FUNCTION F_ParToCsvLine : T_MaxString // convert parameter into csv string (default UDt_Parameter setup)
VAR_INPUT
	stParameter : Udt_Parameter ; 
	nColumn		: UDINT ;
END_VAR
VAR
	sTempString : T_MaxString;
	sTempCsvField : T_MaxString;
END_VAR

CASE nColumn OF 
	0: // number
		sTempString := UDINT_TO_STRING(stParameter.nNumber);
	1: // name
		sTempString := stParameter.sName;
	2: // Type
		sTempString := stParameter.sType;
	3: // discription
		sTempString := stParameter.sDiscription;
	4: // factory
		sTempString := LREAL_TO_STRING(stParameter.fFactory);
	5: // maximum
		sTempString := LREAL_TO_STRING(stParameter.fMaximum);
	6: // minimum
		sTempString := LREAL_TO_STRING(stParameter.fMinimum);
	7: // Unit 
		sTempString := stParameter.sUnit;
	8: // value
		sTempString := LREAL_TO_STRING(stParameter.fValue);
	ELSE
		;
END_CASE

sTempCsvField := STRING_TO_CSVFIELD(sTempString, FALSE);
IF nColumn < 8 THEN 
	sTempCsvField := CONCAT(StempCsvField,';');
ELSE
	sTempCsvField := CONCAT(StempCsvField,'$L');
END_IF

F_ParToCsvLine := sTempCsvField;

END_FUNCTION

(* stored: Version 1.1.0.1, ProductVersion 3.1.4024.6
   POU F_ParToCsvLine: Id {823f7904-d7b6-4ae4-8508-8997ce4f51bf}, SpecialFunc None *)
